FUNCTION_BLOCK F_LINT_TO_LREAL (* Convert LINT to LREAL *)
  (* Standard: 61499-1; Description: Copyright (c) 2023 Martin Erich Jobst This program and the accompanying materials are made available under the terms of the Eclipse Public License 2.0 which is available at https://www.eclipse.org/legal/epl-2.0/ SPDX-License-Identifier: EPL-2.0 *)
  (* Version 1.0, 2023-04-28, Martin Jobst *)
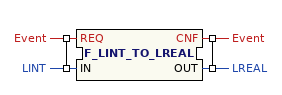
  EVENT_INPUT
    REQ WITH IN; (* Normal Execution Request *)
  END_EVENT
  EVENT_OUTPUT
    CNF WITH OUT; (* Execution Confirmation *)
  END_EVENT
  VAR_INPUT
    IN : LINT;
  END_VAR
  VAR_OUTPUT
    OUT : LREAL;
  END_VAR
  ALGORITHM REQ IN ST:
OUT := LINT_TO_LREAL(IN);
  END_ALGORITHM
END_FUNCTION_BLOCK
